{attribute 'qualified_only'}
VAR_GLOBAL
    //==========================================================
    // HMI通信看门狗配置
    //==========================================================

    // 初次增加程序时保持FALSE。
    // 确认WPF已经能够稳定写入心跳后，再改为TRUE。
    bUseHmiWatchdog : BOOL := FALSE;

    // 超时阈值见GVL_CommunicationConfig；此开关保留WPF现有ADS路径。

END_VAR

(* stored: Version 1.1.0.1, ProductVersion 3.1.4026.20
   GVL GVL_System: Id {e087346e-e6fe-4094-b4e2-6f8a98151646} *)
